Fanuc KAREL source: kb00147.KL

-- PROVISIONAL review KL for V940-1; original PC SHA256 489b912292ca705075ca6e763e9700f634a2ad939b137851d173b417beff35e9
-- Incomplete behavior may be omitted. Consult companion uncertainty JSON. Do not deploy.
PROGRAM KB00147
%NOLOCKGROUP
BEGIN
  -- V9_ZERO_TABLE_METADATA_HINT layout=0002_ascii; no indexed target words; source/name/runtime held
  -- UNRESOLVED_PC offsets 5-14; opcodes 3F,75
  -- UNRESOLVED_PC offsets 19-28; opcodes 3F,75
  -- UNRESOLVED_PC offsets 33-42; opcodes 3F,75
  -- UNRESOLVED_PC offsets 47-54; opcodes 9D,23
  -- UNRESOLVED_PC offsets 59-93; opcodes 27,22,2A,22,2A,22,2A,22,31
  -- UNRESOLVED_PC offsets 98-102; opcodes 7F
END KB00147
